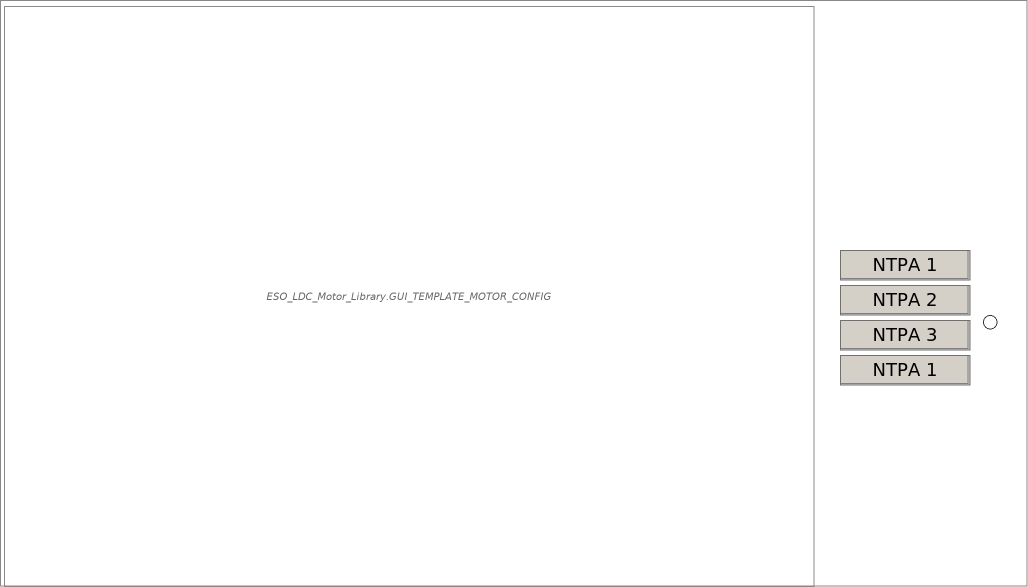
VISUALIZATION GUI_NOTT_TIP_A_CONFIG  // 1028x587
    Frame (4,6 810x581)
        shows ESO_LDC_Motor_Library.GUI_TEMPLATE_MOTOR_CONFIG(m_Instance := MAIN.nott_ics.TipTilt.ptrTipActuatorsA[MAIN.nott_ics.TipTilt.guiTipActuatorsAIndex]^)
    RadioButton (981,252 47x140), variable: MAIN.nott_ics.TipTilt.guiTipActuatorsAIndex-1
        Areas[0]: Text=Radiobutton
        Areas[1]: Text=Radiobutton
    Button (840,250 130x30), "NTPA 1"
        OnMouseClick: execute { MAIN.nott_ics.TipTilt.guiTipActuatorsAIndex := 1; }
    Button (840,285 130x30), "NTPA 2"
        OnMouseClick: execute { MAIN.nott_ics.TipTilt.guiTipActuatorsAIndex := 2; }
    Button (840,320 130x30), "NTPA 3"
        OnMouseClick: execute { MAIN.nott_ics.TipTilt.guiTipActuatorsAIndex := 3; }
    Button (840,355 130x30), "NTPA 1"
        OnMouseClick: execute { MAIN.nott_ics.TipTilt.guiTipActuatorsAIndex := 4; }
END_VISUALIZATION

(* stored: Version 1.1.0.1, ProductVersion 3.1.4024.12
   Visu GUI_NOTT_TIP_A_CONFIG: Id {ffac38f2-9476-49e8-8388-dbccfc68bebc} *)
